// TwinCAT 3 PLC project ScopeTestPLC
// ProgramVersion: 3.1.4024.0
// libraries:
//   Tc2_MC2, * (Beckhoff Automation GmbH)
//   Tc2_Standard, * (Beckhoff Automation GmbH)
//   Tc2_System, * (Beckhoff Automation GmbH)
//   Tc3_Module, * (Beckhoff Automation GmbH)
// project tree:
//   GVLs/ Axes.TcGVL
//   / PlcTask.TcTTO (not stored)
//   POUs/ MAIN.TcPOU (not stored)

// ---- GVLs/Axes.TcGVL
{attribute 'qualified_only'}
VAR_GLOBAL
	Axis1 : AXIS_REF;
END_VAR
